Staubli VAL3: cycle_getLoop.pgx

program cycle_getLoop(bool& x_bLoop[] (dimensions=1))
begin
  // get the loop
  call processList:getLoop(x_bLoop)
end
